(* CoDeSys 2.3 export: FSETK16PUMP.EXP *)

(* POU K16/fSetK16Pump, ST *)
FUNCTION fSetK16Pump : BOOL
VAR_INPUT
	State : BOOL;
	PumpID : USINT;
END_VAR
VAR
END_VAR
	PLC160DO.K16Pump[PumpID] := State;
	(*Включить/Выключить реле насоса*)
END_FUNCTION
